{attribute 'qualified_only'}
VAR_GLOBAL
	 trajectory              :TRAJECTORY;						  //轨迹
END_VAR

(* stored: Version 1.1.0.1, ProductVersion 3.1.4022.10
   GVL TRAJ: Id {b03705c7-8c2d-4274-aa45-be7330ff1fc2} *)
